PROGRAM MAIN
VAR

	fbDrive			  : FB_Drive;
	fbDrive_01		  : FB_Drive;
	fbMotorControl 	  : FB_MotorControl(fbDrive);
	fbMotorControl_01 : FB_MotorControl(fbDrive_01);

	
END_VAR

fbMotorControl();
fbMotorControl_01();

END_PROGRAM

(* stored: Version 1.1.0.1, ProductVersion 3.1.4024.12
   POU MAIN: Id {94995db9-82fb-4583-94ae-a1fd1a7e3270}, SpecialFunc None *)
